TYPE EN_MSG_LIST :
(*************************************************************************************************)
(*  FILENAME:    EN_MSG_LIST.EXP                                                                 *)
(*  PROJECT:     CALMAR PUPLC                                                                    *)
(*  COPYRIGHT:   All rights reserved (c) Wifag//Polytype, Fribourg/Switzerland (2016)            *)
(*  ENVIRONMENT: TwinCAT PLC                                                                     *)
(*  VERSION:     <version>                                                                       *)
(*************************************************************************************************)
(*  DESCRIPTION:                                                                   <description> *)
(*     This block containts the global list for all messages used by `FB_MESSAGE`.               *)
(*                                                                                </description> *)
(*************************************************************************************************)
(
  // start at                       eCStag_MSG_BASE := 10000,
  eC_STAG_CAM_NOTAVAIL                              :=10000,  (*CameraNotAvailable*)
  eC_STAG_CAM_MODE_NOTSUPPORTED                     :=10001,  (*CameraModeNotSupported*)
  eC_STAG_CAM_NOTENGOUGH_TEACH_POINTS               :=10002,  (*CameraNotEnoughTeachPoints*)
  eC_STAG_DEF_SCRIPT_NOT_RUNNING                    :=10003,  (*DeformationScriptNotRunning*)
  eC_STAG_CAM_TEACH_ERROR                           :=10004,  (*CameraTeachError*)
  eC_STAG_IMAGELENGTH_NOT_SUPPORTED                 :=10005,  (*ImageLengthNotSupported*)
  eC_STAG_DEFORMATION_LIMITED                       :=10006   (*DeformationWasLimited (Warning)*)
);
END_TYPE

(* stored: Version 1.1.0.1, ProductVersion 3.1.4024.11
   DUT EN_MSG_LIST: Id {b779ca97-c3e5-47a6-9087-28060a0419c7} *)
